PROGRAM Simulacion
VAR
	vel : REAL := 0.001;

END_VAR

//nuevos ángulos
IF IO.valv_alfa_mas THEN
	IO.alfa_sim:=IO.alfa_sim + vel;
	ELSE IF IO.valv_alfa_menos THEN
		IO.alfa_sim := (IO.alfa_sim - vel);
	END_IF

END_IF

IF IO.valv_beta_mas THEN
	IO.beta_sim:=IO.beta_sim + vel;
	ELSE IF IO.valv_beta_menos THEN
		IO.beta_sim := IO.beta_sim - vel;
	END_IF

END_IF

IO.alfa_sim:=TwoPiCrop(IO.alfa_sim);
IO.beta_sim:=TwoPiCrop(IO.beta_sim);

END_PROGRAM

(* stored: Version 1.1.0.1, ProductVersion 3.1.4024.4
   POU Simulacion: Id {1cb571e3-1b66-4606-979d-4d7d366bccdb}, SpecialFunc None *)
